FUNCTION_BLOCK Interlock (* Basic Function Block Type *)
  (* Standard: 61499-2 *)
  (* Version 0.0, 7/27/2023, vv263, nxtControl GmBH, Template *)
  PACKAGE Main;
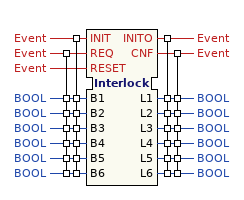
  EVENT_INPUT
    INIT WITH B1, B2, B3, B4, B5, B6; (* Initialization Request *)
    REQ WITH B1, B2, B3, B4, B5, B6; (* Normal Execution Request *)
    RESET;
  END_EVENT
  EVENT_OUTPUT
    INITO WITH L1, L2, L3, L4, L5, L6; (* Initialization Confirm *)
    CNF WITH L1, L2, L3, L4, L5, L6; (* Execution Confirmation *)
  END_EVENT
  VAR_INPUT
    B1 : BOOL; (* Input event qualifier *)
    B2 : BOOL;
    B3 : BOOL;
    B4 : BOOL;
    B5 : BOOL;
    B6 : BOOL;
  END_VAR
  VAR_OUTPUT
    L1 : BOOL; (* Output event qualifier *)
    L2 : BOOL;
    L3 : BOOL;
    L4 : BOOL;
    L5 : BOOL;
    L6 : BOOL;
  END_VAR
  VAR
    NumOn : INT;
    NumLitOn : INT;
  END_VAR
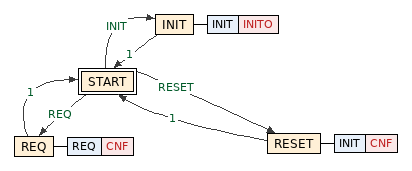
  EC_STATES
    START; (* Initial State *)
    INIT : INIT -> INITO; (* Initialization *)
    REQ : REQ -> CNF; (* Normal execution *)
    RESET : INIT -> CNF;
  END_STATES
  EC_TRANSITIONS
    START TO INIT := INIT;
    INIT TO START := 1;
    START TO REQ := REQ;
    REQ TO START := 1;
    START TO RESET := RESET;
    RESET TO START := 1;
  END_TRANSITIONS
  ALGORITHM INIT IN ST: (* Initialization algorithm *)
L1:=FALSE;
L2:=FALSE;
L3:=FALSE;
L4:=FALSE;
L5:=FALSE;
L6:=FALSE;
  END_ALGORITHM
  ALGORITHM REQ IN ST: (* Normally executed algorithm *)
NumOn:=0;
NumLitOn:=0;
IF B1 THEN NumOn:=NumOn+1; END_IF;
IF B2 THEN NumOn:=NumOn+1; END_IF;
IF B3 THEN NumOn:=NumOn+1; END_IF;
IF B4 THEN NumOn:=NumOn+1; END_IF;
IF B5 THEN NumOn:=NumOn+1; END_IF;
IF B6 THEN NumOn:=NumOn+1; END_IF;

IF L1 THEN NumLitOn:=NumLitOn+1; END_IF;
IF L2 THEN NumLitOn:=NumLitOn+1; END_IF;
IF L3 THEN NumLitOn:=NumLitOn+1; END_IF;
IF L4 THEN NumLitOn:=NumLitOn+1; END_IF;
IF L5 THEN NumLitOn:=NumLitOn+1; END_IF;
IF L6 THEN NumLitOn:=NumLitOn+1; END_IF;

IF (NumOn=1)&(NumLitOn=0) THEN
  L1:=B1;
  L2:=B2;
  L3:=B3;
  L4:=B4;
  L5:=B5;
  L6:=B6;
END_IF;
  END_ALGORITHM
END_FUNCTION_BLOCK
